// TIA Portal project "MachineModeControll_panel3buttons" (V16)

(* hardware
DEVICE "ET 200SP station_1"  ET 200SP-Station
   slot 0: "Rack_0"  Rack  6ES5 710-8MAx1
   slot 1: "PLC_1"  CPU 1510SP-1 PN  6ES7 510-1DJ00-0AB0  V1.8
      slot 32768: "PROFINET interface_1"  X1
         slot 32771: "Port_3"  X1 P3
   slot 2: "Server module_1"  Server module  6ES7 193-6PA00-0AA0  V1.1
      slot 1: "Server module_1"  Server module
   slot 127: "BA 2xRJ45"  BA 2xRJ45  6ES7 193-6AR00-0AA0  V0.0
      slot 32769: "Port_1"  X1 P1  6ES7 193-6AR00-0AA0
      slot 32770: "Port_2"  X1 P2  6ES7 193-6AR00-0AA0
*)

// ===== PLC "PLC_1"  CPU 1510SP-1 PN =====

TYPE "tyPushButtonPanel_Input"
   STRUCT
      bRunPushButton : Bool;
      bStopPushbutton : Bool;
      bResetPushButton : Bool;
   END_STRUCT;
END_TYPE

TYPE "tyMachineModeState"
   STRUCT
      bMachineInStopMode : Bool;
      bMachineInRunMode : Bool;
   END_STRUCT;
END_TYPE

DATA_BLOCK "ModeControll_Panel_DB"   // DB1
{ S7_Optimized_Access := 'TRUE' }
VERSION : 0.1
// stored: InstanceOfName ModeControll_Panel
"ModeControll_Panel"
BEGIN
END_DATA_BLOCK

FUNCTION_BLOCK "ModeControll_Panel"   // FB1, SCL
{ S7_Optimized_Access := 'TRUE' }
VERSION : 0.1
   VAR_INPUT
      MachineControlPanel_Input : "tyPushButtonPanel_Input";
   END_VAR
   VAR_OUTPUT
      MachineModeStateOutput : "tyMachineModeState";
      bGlobalReset : Bool;
   END_VAR
   VAR
      R_Trig_StartPushButton : R_TRIG;
      R_Trig_StopPushButton : R_TRIG;
   END_VAR
BEGIN
   //=============================================================================
   // Dmitri Raihtsaum - Copyright 2023
   // Created By: Dmitri Raihtsaum
   //-----------------------------------------------------------------------------
   // Tested with:   6ES7 510-1DJ00-0AB0
   // Engineering:   TIA Portal V16
   // Functionality: Machine control push buttons logic
   // Date: 09.04.2023
   // Rev 0.1
   //=============================================================================


   //Mapping
   #R_Trig_StartPushButton(CLK:=#MachineControlPanel_Input.bRunPushButton);
   #R_Trig_StopPushButton(CLK := #MachineControlPanel_Input.bStopPushbutton);
   //Protection 
   IF #MachineModeStateOutput.bMachineInStopMode AND #MachineModeStateOutput.bMachineInRunMode THEN
       #MachineModeStateOutput.bMachineInStopMode := TRUE;
       #MachineModeStateOutput.bMachineInRunMode := FALSE;
   END_IF;
   IF NOT #MachineModeStateOutput.bMachineInStopMode AND NOT #MachineModeStateOutput.bMachineInRunMode THEN
       #MachineModeStateOutput.bMachineInStopMode := TRUE;
       #MachineModeStateOutput.bMachineInRunMode := FALSE;
   END_IF;
   //Logic
   //Start button is pressed
   IF #R_Trig_StartPushButton.Q THEN
       #MachineModeStateOutput.bMachineInStopMode := FALSE;
       #MachineModeStateOutput.bMachineInRunMode := TRUE;
   END_IF;
   //Stop button is pressed
   IF #R_Trig_StopPushButton.Q THEN
       #MachineModeStateOutput.bMachineInStopMode := TRUE;
       #MachineModeStateOutput.bMachineInRunMode := FALSE;
   END_IF;
   // Global Reset
   IF #MachineControlPanel_Input.bResetPushButton AND #MachineModeStateOutput.bMachineInStopMode THEN
       #bGlobalReset := TRUE;
   ELSE
       #bGlobalReset := FALSE;
   END_IF;
   //=========================================================================
   //END
   //=========================================================================
END_FUNCTION_BLOCK

ORGANIZATION_BLOCK "Main"   // OB1, LAD, ProgramCycle
TITLE = "Main Program Sweep (Cycle)"
{ S7_Optimized_Access := 'TRUE' }
VERSION : 0.1
   VAR_INPUT
      Initial_Call : Bool;   // Initial call of this OB
      Remanence : Bool;   // =True, if remanent data are available
   END_VAR
BEGIN

REGION Network 1
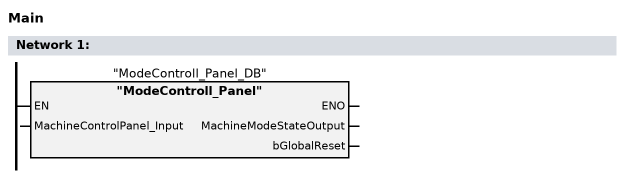
   RUNG wire#powerrail
      "ModeControll_Panel_DB"(MachineControlPanel_Input :=, MachineModeStateOutput =>, bGlobalReset =>)
   END_RUNG
   // the same network as SCL:
   "ModeControll_Panel_DB"();   // "ModeControll_Panel"
END_REGION
END_ORGANIZATION_BLOCK